FUNCTION F_ULINT_ARG : ST_Arg
VAR_INPUT
	nInput : ULINT;
END_VAR
VAR
	stArg : ST_Arg;
	sysVar_Info : __SYSTEM.VAR_INFO;
END_VAR

sysVar_Info 	:= __VARINFO(nInput);
stArg.TypeClass := sysVar_Info.TypeClass;
stArg.pValue 	:= 0;
stArg.diSize 	:= SIZEOF(nInput);
stArg.sValue 	:= TO_STRING(nInput); 
F_ULINT_ARG := stArg;

END_FUNCTION

(* stored: Version 1.1.0.1, ProductVersion 3.1.4024.4
   POU F_ULINT_ARG: Id {b251cae5-0f59-43f8-abfd-1cd942586425}, SpecialFunc None *)
